{attribute 'qualified_only'}
{attribute 'strict'}
{attribute 'to_string'}
TYPE
ST130_Dose_e :
(
    RESET := 0, // Reset

    INIT := 100, // Initialisieren 
    Init_HomeVertical_02,
    Init_Vertical_01Z_at_position,
    Init_HomeVertical_10,
    Init_Vertical_10_Down,
    Init_close_down_feeder,
	Init_clamp_up,

    READY := 999,  // READY to Start, Init Done 
    START := 1000, // Start Zyklisch
  
	open_up_feeder_first, // we ensure that the up clamp is open
	fill_kammer, // we have to wait until the kammer is full 
	
    waitOnMover,     // wait until the mover is there
    MOVER_NEEDED_OP, // Ab here, a mover in position is needed to perform the action

    check_filterhut_presence,      // when the shuttle is at position, we control the presence of the filterhut
	close_up_feeder,
    lift_up_piece_in_workposition, // we lift the piece to place it in the funel
	open_down_feeder,
    load_powder_and_vibrate,
    close_down_feeder,
    release_piece_and_open_up_feeder,
	open_up_feeder,
	clamp_down,
	clamp_up,

    SYNC_MOVER_LEAVE, // MoverMan need to take the mover
    MOVER_FREE_OP,    // here, operation without mover can be done.

    DONE := 8000,  // Ablauf beendet 
    ERROR := 9000, // Fehler 
    _max
);
END_TYPE

(*
back to shuttle
check level NIO Box
*)

(* stored: Version 1.1.0.1, ProductVersion 3.1.4024.6
   EnumerationTextList ST130_Dose_e: Id {851875a3-939a-4324-9ec8-3a0a315cc11b} *)
